Universal Robots PolyScope program: _adminCG-PHomeToConveyor.urp

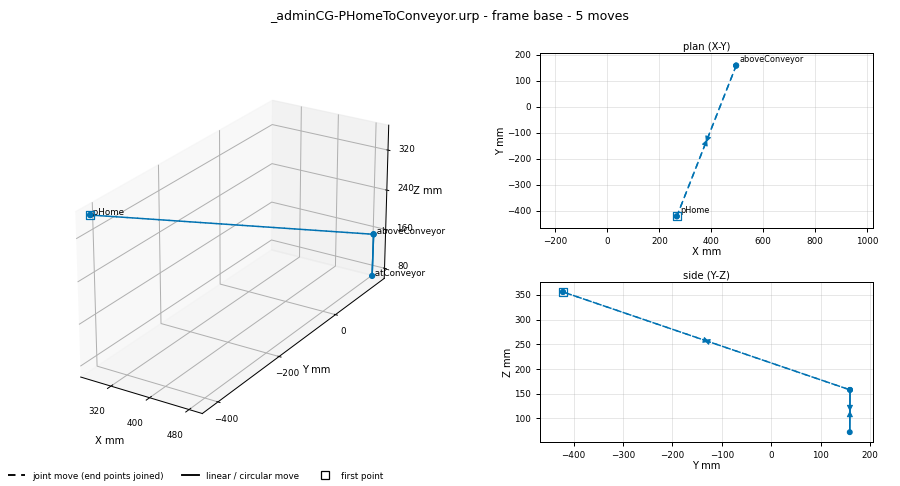
[picture p0: tool path of _adminCG-PHomeToConveyor.urp in frame base, 5 of 5 moves have a stored position in this frame; points joined in program order, loops and branches not executed]
Program _adminCG-PHomeToConveyor (installation=admin directory=/programs/THU_530PM createdIn=3.8.0.61336 lastSavedIn=3.15.8.106339 robotSerialNumber=2015350924)
Calibrated DH parameters: a=[0, -0.425, -0.39225, 0, 0, 0]; d=[0.089159, 0, 0, 0.10915, 0.09465, 0.0823]; alpha=[1.570796, 0, 0, 1.570796, -1.570796, 0]; deltaTheta=[0, 0, 0, 0, 0, 0]
Robot Program (runOnlyOnce=true)
  SuppressedNode
    Set DigitalOutput pin=digital_out[0]; digitalValue=1
  Call _adminLinearIndex1
  MoveJ speed 180 deg/s, acceleration 100 deg/s^2 (useActiveTCP=true)
    Waypoint pHome: TCP in base x=267.077 y=-421.526 z=355.862 mm, rx=1.114 ry=1.1061 rz=0.0051 rad; joints [-45.007, -90.005, -89.993, -90.005, 90, -0.004] deg; flange x=267.08 y=-421.53 z=431.862 mm, rx=1.2021 ry=-2.9025 rz=-0.0001 rad
    Waypoint aboveConveyor: TCP in base x=495.704 y=159.15 z=157.787 mm, rx=0.0126 ry=1.7154 rz=1.2129 rad; joints [29.849, -99.883, -109.293, -61.157, 90.169, -14.961] deg; flange x=496.198 y=159.176 z=233.785 mm, rx=2.8978 ry=-1.206 rz=-0.0092 rad
  MoveL speed 250 mm/s, acceleration 1200 mm/s^2 (useActiveTCP=true) feature=Base
    Waypoint atConveyor: TCP in base x=495.183 y=158.608 z=72.185 mm, rx=0.0126 ry=1.7154 rz=1.2129 rad; joints [29.826, -107.098, -115.272, -47.963, 90.167, -14.983] deg; flange x=495.677 y=158.635 z=148.183 mm, rx=2.8978 ry=-1.206 rz=-0.0092 rad
    Set DigitalOutput pin=digital_out[0]; digitalValue=0
    Wait Sleep waitTime=1
    Waypoint aboveConveyor: TCP in base x=495.704 y=159.15 z=157.787 mm, rx=0.0126 ry=1.7154 rz=1.2129 rad; joints [29.849, -99.883, -109.293, -61.157, 90.169, -14.961] deg; flange x=496.198 y=159.176 z=233.785 mm, rx=2.8978 ry=-1.206 rz=-0.0092 rad
  MoveJ speed 180 deg/s, acceleration 100 deg/s^2 (useActiveTCP=true)
    Waypoint phome: TCP in base x=267.106 y=-421.453 z=355.828 mm, rx=1.114 ry=1.1062 rz=0.0052 rad; joints [-45, -90.001, -90.002, -90.005, 90.003, -0.002] deg; flange x=267.11 y=-421.463 z=431.828 mm, rx=1.2023 ry=-2.9024 rz=-0.0002 rad
SubProgram  [hidden by the author, left out]
SubProgram _adminLinearIndex1 [hidden by the author, left out]
